// SIMATIC S7-200 project (STEP 7-Micro/WIN), CPU 221 REL 01.10

SYMBOL_TABLE USER1
start            I0.0
estop            I0.1
s1               I0.2     // cam bien hop
s2               I0.3     // cam bien tao
BTH              Q0.0     // bang tai hop
BTT              Q0.1     // bang tai tao
END_SYMBOL_TABLE

ORGANIZATION_BLOCK MAIN:OB1
TITLE=PROGRAM COMMENTS
BEGIN
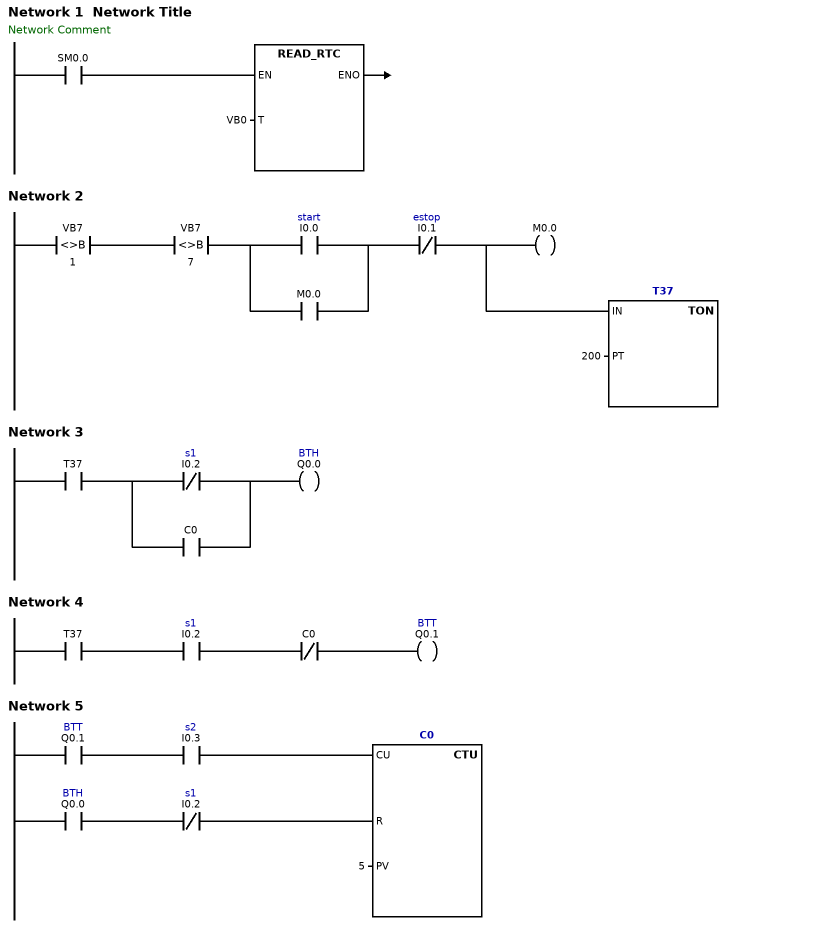
Network 1 // Network Title
// Network Comment
LD     SM0.0
TODR   VB0
Network 2
LDB<>  VB7, 1
AB<>   VB7, 7
LD     start:I0.0
O      M0.0
ALD
AN     estop:I0.1
=      M0.0
TON    T37, 200
Network 3
LD     T37
LDN    s1:I0.2
O      C0
ALD
=      BTH:Q0.0
Network 4
LD     T37
A      s1:I0.2
AN     C0
=      BTT:Q0.1
Network 5
LD     BTT:Q0.1
A      s2:I0.3
LD     BTH:Q0.0
AN     s1:I0.2
CTU    C0, 5
END_ORGANIZATION_BLOCK
